// TIA Portal V16 export
// export: Created 2021-08-30T13:11:27.0142557Z, ExportSetting WithDefaults, DisplayName Totally Integrated Automation Portal, DisplayVersion V16 Update 3, DisplayName TIA Portal Version Control Interface, DisplayVersion V16 Update 2, DisplayName TIA Portal Openness, DisplayVersion V16 Update 3, DisplayName TIA Portal Teamcenter Gateway, DisplayVersion V16, DisplayName STEP 7 Professional, DisplayVersion V16 Update 3, DisplayName STEP 7 Safety, DisplayVersion V16, DisplayName WinCC Advanced, DisplayVersion V16 Update 3
FUNCTION_BLOCK "DPumpCntr"   // FB70, LAD
{ S7_Optimized_Access := 'FALSE' }
VERSION : 0.1
// #ST:
// номер бита, часло десятичное
//  0  - стоп 
// 0 1 - работа
// 1 2 - запуск
// 2 4 - остановка
// 3 8 - сервисный режим
// 4 16 - ошибка Пуска
// 5 32 - ошибка Стопа
// 6 64 - ошибка питания
// 7 128 - ошибка частотника (дозатора)
// 8 256 - Блокировка внешняя
// 9 - 512 - нажат аварийный стоп
// 10 -1024 - сборная авария
// 11 2048
// 12 4096
// 13 8192
// 14 16384 
// 15 32768 - режим 0-ручной, 1-авто
// 
// 
// 
// показывать кнопки ручного управления
// stored: AutoNumber false, IsIECCheckEnabled false, SetENOAutomatically false, UDAEnableTagReadback false
   VAR_INPUT
      power : Bool;   // питание устройства
      run : Bool;
      emrStop : Bool;   // Авариный стоп 0-авария, 1-ок
      alarmFC : Bool;   // 1-авария
      Ack : Bool;   // Сброс Аварий
      FE : Real;
   END_VAR
   VAR_OUTPUT
      qStart : Bool;
      pqw : Int;
   END_VAR
   VAR_IN_OUT
      dev : "DPump";
      prop : "PropDosing";
   END_VAR
   VAR DB_SPECIFIC
      ErrOC : Bool;   // Признак аварии по закрытию или открытию
      ErrPower : Bool;   // Признак аварии питания
      ErrDis : Bool;   // Признак внешней блокировки
      qON : Bool;   // Выход для управления механизмом
      tmrClosing { S7_SetPoint := 'True'} : TON_TIME;
      tmrOpening { S7_SetPoint := 'True'} : TON_TIME;
      closed : Bool;
      opened : Bool;
      closing : Bool;
      opening : Bool;
      errStart : Bool;
      errStop : Bool;
      errEmrStop : Bool;
      errAlarmFc : Bool;
      errService : Bool;
      tStart : Time;
      tStop : Time;
   END_VAR
   VAR
      ServiceEventHandler { S7_SetPoint := 'True'} : "DevAckSingleAlarm";
      PowerEventHandler { S7_SetPoint := 'True'} : "DevAckSingleAlarm";
      DevAlarmEventHandler { S7_SetPoint := 'True'} : "DevAckSingleAlarm";
      DisEventHandler { S7_SetPoint := 'True'} : "DevAckSingleAlarm";
      EmrStopEventHandler { S7_SetPoint := 'True'} : "DevAckSingleAlarm";
      BadStartEventHandler { S7_SetPoint := 'True'} : "DevAckSingleAlarm";
      BadStopEventHandler { S7_SetPoint := 'True'} : "DevAckSingleAlarm";
   END_VAR
BEGIN

REGION Network 1: Сброс состояния
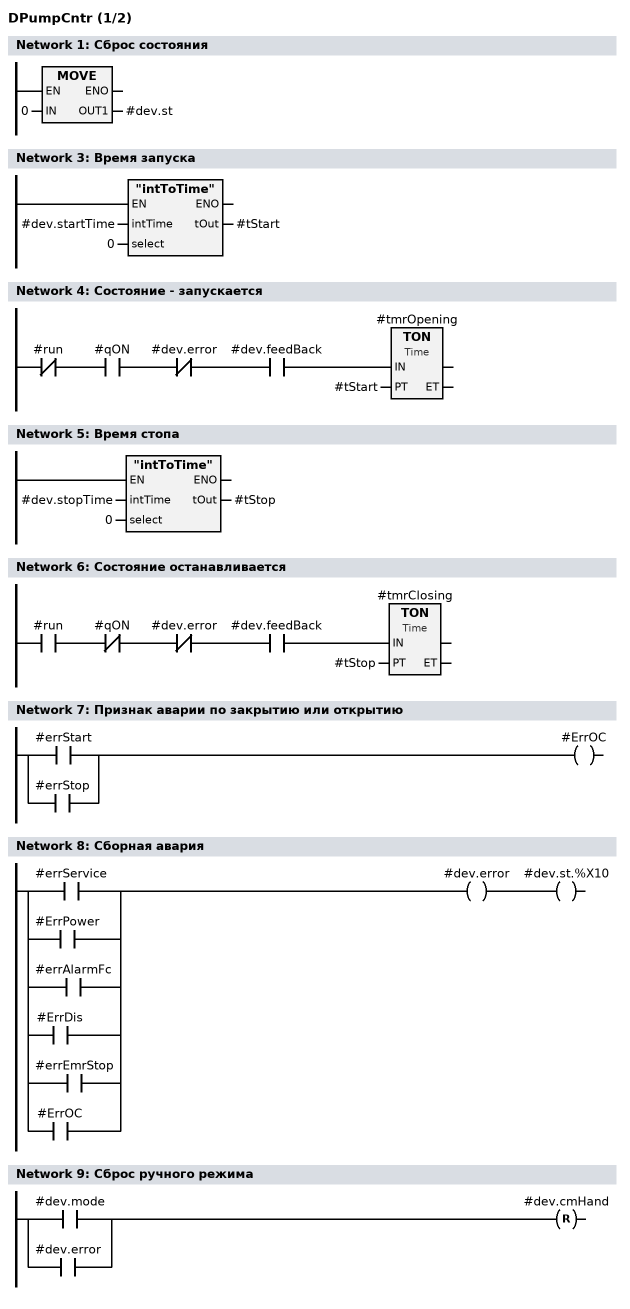
   RUNG wire#powerrail
      { S7_GenerateENO := "TRUE" } Move(in := 0, out1 => #dev.st)
   END_RUNG
   // the same network as SCL:
   #dev.st := 0;
END_REGION

REGION Network 2 (SCL): Event handlers
   #ServiceEventHandler(alarmSignal := #dev.service,
                        ack := #Ack,
                        ackBit := #dev.ack.%X3,
                        stateBit := #dev.st.%X3,
                        alarmTag := #errService);
   #BadStartEventHandler(alarmSignal:=#tmrOpening.Q,
                         ack:=#Ack,
                         ackBit:=#dev.ack.%X4,
                         stateBit:=#dev.st.%X4,
                         alarmTag:=#errStart);
   #BadStopEventHandler(alarmSignal:=#tmrClosing.Q,
                        ack:=#Ack,
                        ackBit:=#dev.ack.%X5,
                        stateBit:=#dev.ack.%X5,
                        alarmTag:=#errStop);
   #PowerEventHandler(alarmSignal := #power,
                      ack := #Ack,
                      ackBit := #dev.ack.%X6,
                      stateBit := #dev.st.%X6,
                      alarmTag := #ErrPower);
   #DevAlarmEventHandler(alarmSignal := #alarmFC,
                         ack := #Ack,
                         ackBit := #dev.ack.%X7,
                         stateBit := #dev.st.%X7,
                         alarmTag := #errAlarmFc);
   #DisEventHandler(alarmSignal := #dev.block,
                    ack := #Ack,
                    ackBit := #dev.ack.%X8,
                    stateBit := #dev.st.%X8,
                    alarmTag := #ErrDis);
   #EmrStopEventHandler(alarmSignal := #emrStop,
                        ack := #Ack,
                        ackBit := #dev.ack.%X9,
                        stateBit := #dev.st.%X9,
                        alarmTag := #errEmrStop);
END_REGION

REGION Network 3: Время запуска
   RUNG wire#powerrail
      "intToTime"(intTime := #dev.startTime, select := 0, tOut => #tStart)
   END_RUNG
   // the same network as SCL:
   "intToTime"(intTime := #dev.startTime, select := 0, tOut => #tStart);
END_REGION

REGION Network 4: Состояние - запускается
   RUNG wire#powerrail
      I_Contact( #run )
      Contact( #qON )
      I_Contact( #dev.error )
      Contact( #dev.feedBack )
      { S7_Templates := "time_type := Time" } #tmrOpening.TON(pt := #tStart, et =>)
   END_RUNG
   // the same network as SCL:
   #tmrOpening(IN := NOT #run AND #qON AND NOT #dev.error AND #dev.feedBack, PT := #tStart);   // TON
END_REGION

REGION Network 5: Время стопа
   RUNG wire#powerrail
      "intToTime"(intTime := #dev.stopTime, select := 0, tOut => #tStop)
   END_RUNG
   // the same network as SCL:
   "intToTime"(intTime := #dev.stopTime, select := 0, tOut => #tStop);
END_REGION

REGION Network 6: Состояние останавливается
   RUNG wire#powerrail
      Contact( #run )
      I_Contact( #qON )
      I_Contact( #dev.error )
      Contact( #dev.feedBack )
      { S7_Templates := "time_type := Time" } #tmrClosing.TON(pt := #tStop, et =>)
   END_RUNG
   // the same network as SCL:
   #tmrClosing(IN := #run AND NOT #qON AND NOT #dev.error AND #dev.feedBack, PT := #tStop);   // TON
END_REGION

REGION Network 7: Признак аварии по закрытию или открытию
   RUNG wire#powerrail
      Contact( #errStart )
      wire#w1
      Coil( #ErrOC )
   END_RUNG
   RUNG wire#powerrail
      Contact( #errStop )
   END_RUNG wire#w1
   // the same network as SCL:
   #ErrOC := #errStart OR #errStop;
END_REGION

REGION Network 8: Сборная авария
   RUNG wire#powerrail
      Contact( #errService )
      wire#w1
      Coil( #dev.error )
      Coil( #dev.st.%X10 )
   END_RUNG
   RUNG wire#powerrail
      Contact( #ErrPower )
   END_RUNG wire#w1
   RUNG wire#powerrail
      Contact( #errAlarmFc )
   END_RUNG wire#w1
   RUNG wire#powerrail
      Contact( #ErrDis )
   END_RUNG wire#w1
   RUNG wire#powerrail
      Contact( #errEmrStop )
   END_RUNG wire#w1
   RUNG wire#powerrail
      Contact( #ErrOC )
   END_RUNG wire#w1
   // the same network as SCL:
   #dev.error := #errService OR #ErrPower OR #errAlarmFc OR #ErrDis OR #errEmrStop OR #ErrOC;
   #dev.st.%X10 := #dev.error;
END_REGION

REGION Network 9: Сброс ручного режима
   RUNG wire#powerrail
      Contact( #dev.mode )
      wire#w1
      R_Coil( #dev.cmHand )
   END_RUNG
   RUNG wire#powerrail
      Contact( #dev.error )
   END_RUNG wire#w1
   // the same network as SCL:
   IF #dev.mode OR #dev.error THEN #dev.cmHand := FALSE; END_IF;
END_REGION

REGION Network 10: Сброс авто режима
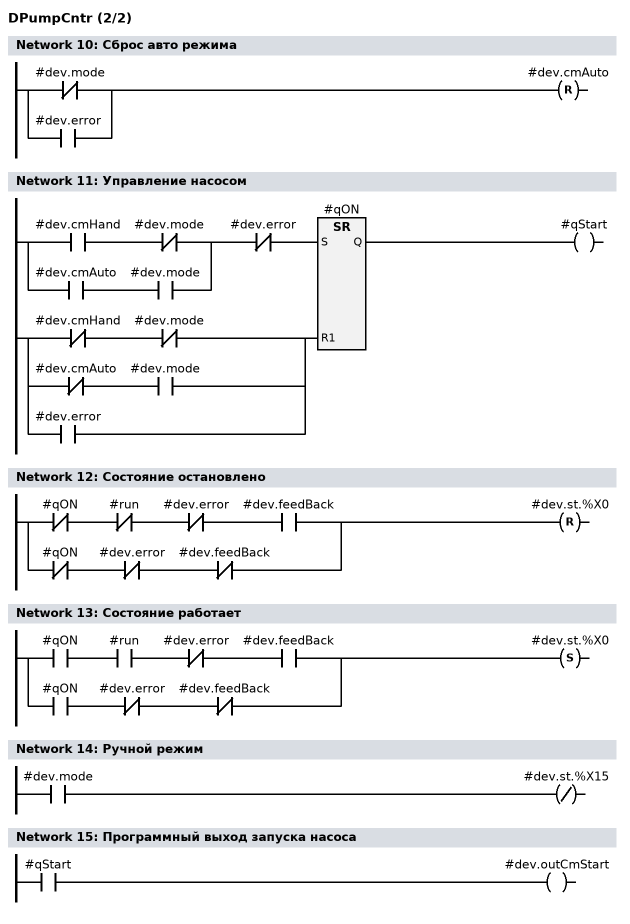
   RUNG wire#powerrail
      I_Contact( #dev.mode )
      wire#w1
      R_Coil( #dev.cmAuto )
   END_RUNG
   RUNG wire#powerrail
      Contact( #dev.error )
   END_RUNG wire#w1
   // the same network as SCL:
   IF NOT #dev.mode OR #dev.error THEN #dev.cmAuto := FALSE; END_IF;
END_REGION

REGION Network 11: Управление насосом
   RUNG wire#powerrail
      Contact( #dev.cmHand )
      I_Contact( #dev.mode )
      wire#w1
      I_Contact( #dev.error )
      S_SR(operand := #qON, r1 := wire#w2)
      Coil( #qStart )
   END_RUNG
   RUNG wire#powerrail
      Contact( #dev.cmAuto )
      Contact( #dev.mode )
   END_RUNG wire#w1
   RUNG wire#powerrail
      I_Contact( #dev.cmHand )
      I_Contact( #dev.mode )
   END_RUNG wire#w2
   RUNG wire#powerrail
      I_Contact( #dev.cmAuto )
      Contact( #dev.mode )
   END_RUNG wire#w2
   RUNG wire#powerrail
      Contact( #dev.error )
   END_RUNG wire#w2
   // the same network as SCL:
   IF ((#dev.cmHand AND NOT #dev.mode) OR (#dev.cmAuto AND #dev.mode)) AND NOT #dev.error THEN
       #qON := TRUE;   // SR flip-flop
   END_IF;
   IF (NOT #dev.cmHand AND NOT #dev.mode) OR (NOT #dev.cmAuto AND #dev.mode) OR #dev.error THEN
       #qON := FALSE;
   END_IF;
   #qStart := #qON;
END_REGION

REGION Network 12: Состояние остановлено
   RUNG wire#powerrail
      I_Contact( #qON )
      I_Contact( #run )
      I_Contact( #dev.error )
      Contact( #dev.feedBack )
      wire#w1
      R_Coil( #dev.st.%X0 )
   END_RUNG
   RUNG wire#powerrail
      I_Contact( #qON )
      I_Contact( #dev.error )
      I_Contact( #dev.feedBack )
   END_RUNG wire#w1
   // the same network as SCL:
   IF (NOT #qON AND NOT #run AND NOT #dev.error AND #dev.feedBack) OR (NOT #qON AND NOT #dev.error AND NOT #dev.feedBack) THEN
       #dev.st.%X0 := FALSE;
   END_IF;
END_REGION

REGION Network 13: Состояние работает
   RUNG wire#powerrail
      Contact( #qON )
      Contact( #run )
      I_Contact( #dev.error )
      Contact( #dev.feedBack )
      wire#w1
      S_Coil( #dev.st.%X0 )
   END_RUNG
   RUNG wire#powerrail
      Contact( #qON )
      I_Contact( #dev.error )
      I_Contact( #dev.feedBack )
   END_RUNG wire#w1
   // the same network as SCL:
   IF (#qON AND #run AND NOT #dev.error AND #dev.feedBack) OR (#qON AND NOT #dev.error AND NOT #dev.feedBack) THEN
       #dev.st.%X0 := TRUE;
   END_IF;
END_REGION

REGION Network 14: Ручной режим
   RUNG wire#powerrail
      Contact( #dev.mode )
      I_Coil( #dev.st.%X15 )
   END_RUNG
   // the same network as SCL:
   #dev.st.%X15 := NOT #dev.mode;
END_REGION

REGION Network 15: Программный выход запуска насоса
   RUNG wire#powerrail
      Contact( #qStart )
      Coil( #dev.outCmStart )
   END_RUNG
   // the same network as SCL:
   #dev.outCmStart := #qStart;
END_REGION

REGION Network 16 (SCL): Prop dossing
   //дозирование пропорционально расходу

   //производителньность л/ч

   IF #dev.mode AND #dev.cmAuto THEN
       //KVA
       IF #prop.enableFix THEN
           IF #prop.fixSP > 100 THEN
               #prop.fixSP := 100;
           END_IF;
           IF #prop.fixSP < 0 THEN
               #prop.fixSP := 0;
           END_IF;
           #prop.outLPH := (#prop.max * #prop.fixSP) / 100;
           //
           // #prop.outLPH := #prop.fixSP;
       ELSE
           IF #prop.density > 0 THEN
               #prop.outLPH := #FE * #prop.spAuto / (#prop.density * 1000.0);
           ELSE
               #prop.outLPH := 0;
           END_IF;

           //запрет дозирования если расход меньше заданного
           IF #FE < #prop.minFE THEN
               #prop.outLPH := 0.0;
           END_IF;
       END_IF;
   END_IF;
   IF NOT #dev.mode AND #dev.cmHand THEN
       #prop.outLPH := #prop.spHand;
   END_IF;

   //запрет дозирования
   IF NOT #dev.cmHand AND NOT #dev.cmAuto THEN
       #prop.outLPH := 0.0;
   END_IF;

   IF #prop.outLPH > #prop.max THEN
       #prop.outLPH := #prop.max;
   END_IF;

   //расчет PQW
   IF #prop.max > 0 THEN
       #pqw := REAL_TO_INT(#prop.outLPH * 27648.0 / #prop.max);
   ELSE
       #pqw := 0;
   END_IF;

   //ограничение выхода
   IF #pqw < 0 THEN
       #pqw := 0;
   END_IF;
   IF #pqw > 27648 THEN
       #pqw := 27648;
   END_IF;
   //расчет тока
   #prop.outmA := 4.0 + INT_TO_REAL(#pqw) * 16.0 / 27648.0;
   #prop.outSP := INT_TO_REAL(#pqw) * 100.0 / 27648.0;
   #prop.FE := #FE;
END_REGION
END_FUNCTION_BLOCK
